{attribute 'linkalways'} 
{attribute 'no_explicit_call' := 'This FB is a CLASS and must be accessed using methods or properties'}
{attribute 'enable_dynamic_creation'}
FUNCTION_BLOCK Node_F_VN_AddToContainerElements_TcVnRotatedRectangle EXTENDS VisionNode
VAR
    stValue : _TcVnRotatedRectangle;
    ipContainer : _ITcVnContainer;
    hrPrev : _HRESULT(S_OK);
    hresult : _HRESULT(S_OK);
END_VAR

METHOD PUBLIC  Clone : I_Node
VAR
    pNode : POINTER TO Node_F_VN_AddToContainerElements_TcVnRotatedRectangle;
END_VAR
pNode := __NEW(Node_F_VN_AddToContainerElements_TcVnRotatedRectangle);
Clone := pNode^;
END_METHOD

METHOD FB_init : BOOL
VAR_INPUT
    bInitRetains : BOOL; // if TRUE, the retain variables are initialized (warm start / cold start)
    bInCopyCode : BOOL;  // if TRUE, the instance afterwards gets moved into the copy code (online change)
END_VAR
AddInput('stValue', stValue);
AddInput('ipContainer', ipContainer);
AddInput('hrPrev', hrPrev);
AddOutput('ipContainer', ipContainer);
AddOutput('hresult',hresult);
END_METHOD

METHOD PROTECTED OnExecute
hresult.Value := F_VN_AddToContainerElements_TcVnRotatedRectangle(
    stValue := stValue.Value,
    ipContainer := ipContainer.Value,
    hrPrev:= hrPrev.Value);
END_METHOD

METHOD PUBLIC PreExecutionCheck
VAR_INPUT
    Check : I_PreExecutionChecks;
END_VAR
Check.IsTrue(ipContainer.IsValid, 'ipContainer must be a valid container');
Check.IsTrue(ipContainer.IsType(TC_GLOBAL_CONST_LIST.ContainerType_Vector_TcVnRotatedRectangle), 'ipContainer contains incorrect type');
END_METHOD

END_FUNCTION_BLOCK

(* stored: Version 1.1.0.1, ProductVersion 3.1.4026.13
   POU Node_F_VN_AddToContainerElements_TcVnRotatedRectangle: Id {c1759959-f282-03b5-073f-d9b2c56f986f}, SpecialFunc None
   Folder Constructor: Id {52f43bc7-b9c1-0658-1f41-ca7d53fdf788}
   Method Clone: Id {d939e7ee-9ebc-0aab-1742-c067b903492e}
   Method FB_init: Id {f3dc24c0-5798-0456-246f-0c8cb2757aad}
   Method OnExecute: Id {d2f24ab2-d233-0ec1-2362-95ecadcba636}
   Method PreExecutionCheck: Id {571e7a61-43ac-0c54-0e84-df19cd8efed0} *)
